% RSLogix 500 project Digital Filling Station.RSS, saved by version 8.30.00.16 %
PROJECT "UNTITLED"    % processor: Bul.1763 MicroLogix 1100 Series B %

PROGRAM FILES
  LAD 2   4 rungs
  LAD 3 "IO"  8 rungs
  LAD 4 "CTRL"  6 rungs
  LAD 5 "CYCLE"  5 rungs

DATA FILES
  O0 OUTPUT  4 elements
  I1 INPUT  6 elements
  S2 STATUS  66 elements
  B3 BINARY  1 elements
  T4 TIMER  1 elements
  C5 COUNTER  1 elements
  R6 CONTROL  1 elements
  N7 INTEGER  1 elements
  F8 FLOAT  1 elements

LADDER 2
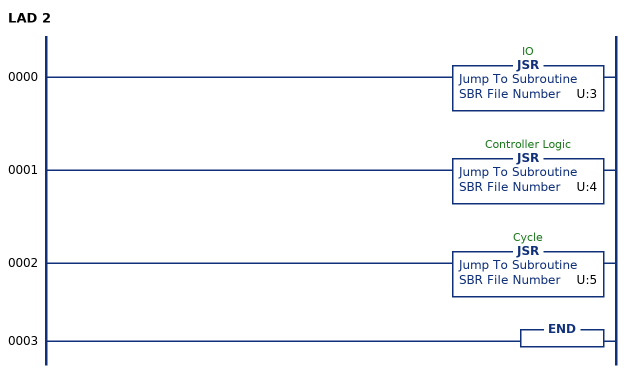
% Rung: 0 %
SOR JSR U:3 EOR
%   U:3  "IO" %
% Rung: 1 %
SOR JSR U:4 EOR
%   U:4  "Controller Logic" %
% Rung: 2 %
SOR JSR U:5 EOR
%   U:5  "Cycle" %
% Rung: 3 %
SOR END EOR

LADDER 3 "IO"
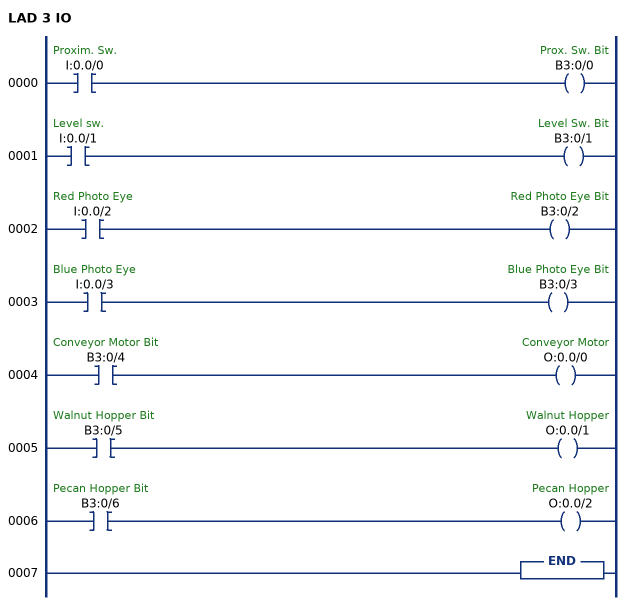
% Rung: 0 %
SOR XIC I:0.0/0 OTE B3:0/0 EOR
%   I:0.0/0  "Proxim. Sw." %
%   B3:0/0  "Prox. Sw. Bit" %
% Rung: 1 %
SOR XIC I:0.0/1 OTE B3:0/1 EOR
%   I:0.0/1  "Level sw." %
%   B3:0/1  "Level Sw. Bit" %
% Rung: 2 %
SOR XIC I:0.0/2 OTE B3:0/2 EOR
%   I:0.0/2  "Red Photo Eye" %
%   B3:0/2  "Red Photo Eye Bit" %
% Rung: 3 %
SOR XIC I:0.0/3 OTE B3:0/3 EOR
%   I:0.0/3  "Blue Photo Eye" %
%   B3:0/3  "Blue Photo Eye Bit" %
% Rung: 4 %
SOR XIC B3:0/4 OTE O:0.0/0 EOR
%   B3:0/4  "Conveyor Motor Bit" %
%   O:0.0/0  "Conveyor Motor" %
% Rung: 5 %
SOR XIC B3:0/5 OTE O:0.0/1 EOR
%   B3:0/5  "Walnut Hopper Bit" %
%   O:0.0/1  "Walnut Hopper" %
% Rung: 6 %
SOR XIC B3:0/6 OTE O:0.0/2 EOR
%   B3:0/6  "Pecan Hopper Bit" %
%   O:0.0/2  "Pecan Hopper" %
% Rung: 7 %
SOR END EOR

LADDER 4 "CTRL"
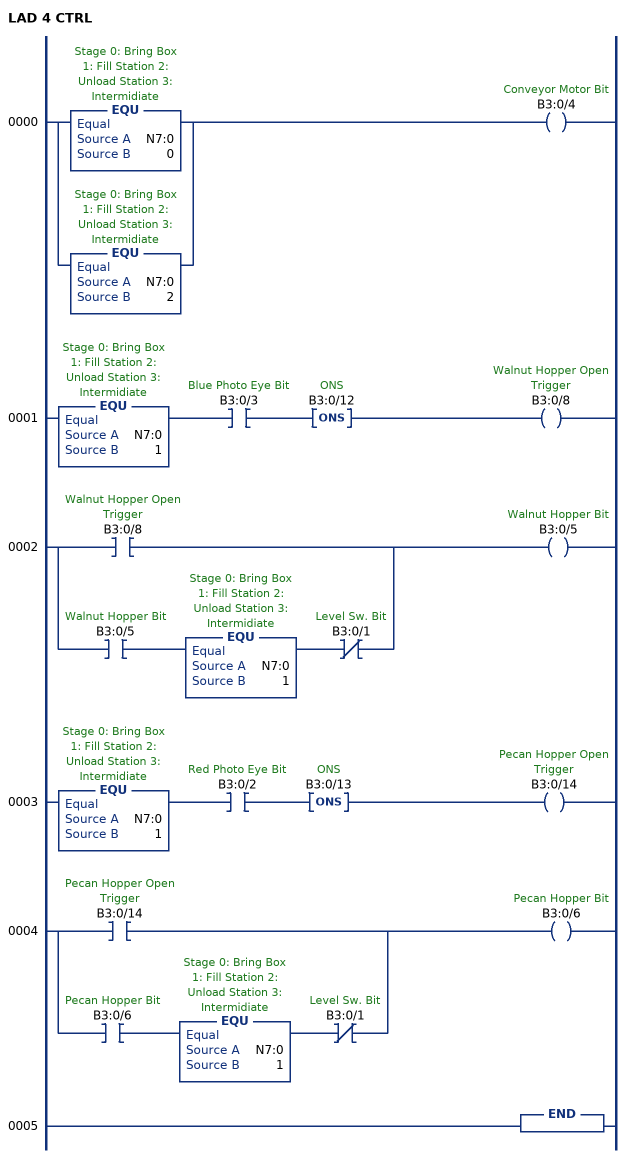
% Rung: 0 %
SOR BST EQU N7:0 0 NXB EQU N7:0 2 BND OTE B3:0/4 EOR
%   N7:0  "Stage 0: Bring Box 1: Fill Station 2: Unload Station 3: Intermidiate" %
%   B3:0/4  "Conveyor Motor Bit" %
% Rung: 1 %
SOR EQU N7:0 1 XIC B3:0/3 ONS B3:0/12 OTE B3:0/8 EOR
%   N7:0  "Stage 0: Bring Box 1: Fill Station 2: Unload Station 3: Intermidiate" %
%   B3:0/3  "Blue Photo Eye Bit" %
%   B3:0/12  "ONS" %
%   B3:0/8  "Walnut Hopper Open Trigger" %
% Rung: 2 %
SOR BST XIC B3:0/8 NXB XIC B3:0/5 EQU N7:0 1 XIO B3:0/1 BND OTE B3:0/5 EOR
%   B3:0/8  "Walnut Hopper Open Trigger" %
%   B3:0/5  "Walnut Hopper Bit" %
%   N7:0  "Stage 0: Bring Box 1: Fill Station 2: Unload Station 3: Intermidiate" %
%   B3:0/1  "Level Sw. Bit" %
% Rung: 3 %
SOR EQU N7:0 1 XIC B3:0/2 ONS B3:0/13 OTE B3:0/14 EOR
%   N7:0  "Stage 0: Bring Box 1: Fill Station 2: Unload Station 3: Intermidiate" %
%   B3:0/2  "Red Photo Eye Bit" %
%   B3:0/13  "ONS" %
%   B3:0/14  "Pecan Hopper Open Trigger" %
% Rung: 4 %
SOR BST XIC B3:0/14 NXB XIC B3:0/6 EQU N7:0 1 XIO B3:0/1 BND OTE B3:0/6 EOR
%   B3:0/14  "Pecan Hopper Open Trigger" %
%   B3:0/6  "Pecan Hopper Bit" %
%   N7:0  "Stage 0: Bring Box 1: Fill Station 2: Unload Station 3: Intermidiate" %
%   B3:0/1  "Level Sw. Bit" %
% Rung: 5 %
SOR END EOR

LADDER 5 "CYCLE"
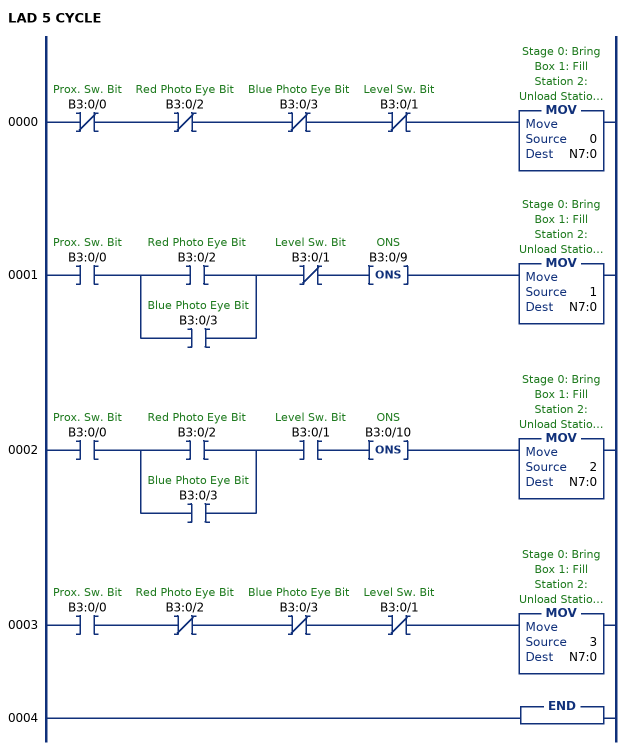
% Rung: 0 %
SOR XIO B3:0/0 XIO B3:0/2 XIO B3:0/3 XIO B3:0/1 MOV 0 N7:0 EOR
%   B3:0/0  "Prox. Sw. Bit" %
%   B3:0/2  "Red Photo Eye Bit" %
%   B3:0/3  "Blue Photo Eye Bit" %
%   B3:0/1  "Level Sw. Bit" %
%   N7:0  "Stage 0: Bring Box 1: Fill Station 2: Unload Station 3: Intermidiate" %
% Rung: 1 %
SOR XIC B3:0/0 BST XIC B3:0/2 NXB XIC B3:0/3 BND XIO B3:0/1 ONS B3:0/9 MOV 1 N7:0 EOR
%   B3:0/0  "Prox. Sw. Bit" %
%   B3:0/2  "Red Photo Eye Bit" %
%   B3:0/3  "Blue Photo Eye Bit" %
%   B3:0/1  "Level Sw. Bit" %
%   B3:0/9  "ONS" %
%   N7:0  "Stage 0: Bring Box 1: Fill Station 2: Unload Station 3: Intermidiate" %
% Rung: 2 %
SOR XIC B3:0/0 BST XIC B3:0/2 NXB XIC B3:0/3 BND XIC B3:0/1 ONS B3:0/10 MOV 2 N7:0 EOR
%   B3:0/0  "Prox. Sw. Bit" %
%   B3:0/2  "Red Photo Eye Bit" %
%   B3:0/3  "Blue Photo Eye Bit" %
%   B3:0/1  "Level Sw. Bit" %
%   B3:0/10  "ONS" %
%   N7:0  "Stage 0: Bring Box 1: Fill Station 2: Unload Station 3: Intermidiate" %
% Rung: 3 %
SOR XIC B3:0/0 XIO B3:0/2 XIO B3:0/3 XIO B3:0/1 MOV 3 N7:0 EOR
%   B3:0/0  "Prox. Sw. Bit" %
%   B3:0/2  "Red Photo Eye Bit" %
%   B3:0/3  "Blue Photo Eye Bit" %
%   B3:0/1  "Level Sw. Bit" %
%   N7:0  "Stage 0: Bring Box 1: Fill Station 2: Unload Station 3: Intermidiate" %
% Rung: 4 %
SOR END EOR

OTHER DOCUMENTED ADDRESSES
  JSR  
  PFILE:4  "CTRL"

DATA TABLE (non-zero values as saved)
DATA B3
% B3:0 % 0X0001
DATA N7
% N7:0 % 3
